(* CoDeSys 2.3.9.41 project: plastic_molding.pro *)
(* Libraries: Standard.lib 4.10.05 11:14:46, IecSfc.lib 13.4.06 15:51:28, SYSLIBCALLBACK.LIB 26.9.08 16:43:52 *)

(* Task configuration *)
TASK NewTask (PRIORITY := 1); (* freewheeling *)
	VIS_PRG();
	PLC_PRG();
END_TASK

(* Global variable list: Global_Variables *)
VAR_GLOBAL (* 11 inputs and 20 outputs *)
	(* Inputs *)
		(* Push buttons: *)
		StartPB: BOOL;
		StopPB: BOOL;
		InterruptPB: BOOL;

		(* Sensors: *)
		Weight0S: BOOL;
		Weight1S: BOOL;
		ClosedDamperS: BOOL;
		OpenedDamperS: BOOL;
		TareS: BOOL;
		UpperTempS: BOOL;
		BottomTempS: BOOL;
		WorkingTempS: BOOL;

	(* Outputs *)
		(* Actuators / Lamps *)
		StartFeed: BOOL;
		OpenValve: BOOL;
		RunConveyor: BOOL;
		OpenDamper: BOOL;
		CloseDamper: BOOL;
		TurnOnHeater: BOOL;

		(* States / Lamps *)
		SystemIsOn: BOOL;
		Stopping: BOOL;
		Melting: BOOL;
		NoFeed: BOOL;
		BrokenHeater: BOOL;
		NoTare: BOOL;

		(* Lamps *)
		EmptyDispenserLmp: BOOL;
		FullDispenserLmp: BOOL;
		TrippedTareSLmp: BOOL;
		OpenedDamperLmp: BOOL;
		ClosedDamperLmp: BOOL;
		UpperTempLmp: BOOL;
		BottomTempLmp: BOOL;
		WorkingTempLmp: BOOL;

	(* Timers are in global variables temporarily for convenience. *)
	FeederTmr: TON := (PT := T#7s);  (* Wating for feeding *)
	HeaterTmr: TON := (PT := T#12s); (* Wating for heating *)
	TareTmr: TON := (PT := T#7s); (* Waiting for tare *)
	MeltingTmr: TON := (PT := T#7s); (* Wating for melting *)
END_VAR

(* POU VIS_PRG, ST *)
PROGRAM VIS_PRG
VAR
	(* Buttons *)
	FillFeedingTowerBtn: BOOL;
	FreeFeedingTowerBtn: BOOL;
	HeaterBreakingToggleBtn: BOOL;
	FirstTareBtn, SecondTareBtn, ThirdTareBtn, FourthTareBtn  : BOOL;
	(* Others *)
	RawPlasticsVlm, _RawPlasticsVlm: INT;   (* Volume *)
	PlasticsPortionVlm,   _PlasticsPortionVlm: INT;  (* Volume *)
	PlasticsPortionClr:      DWORD;            (* Color *)
	Red,  _Red: INT;             (* Red component of the portion color *)
	(* Heater *)
	HeaterClr: DWORD:=16#00_FF_FF_FF;
	HeaterRed, _HeaterRed: BYTE;         (* Red component of the heater color  *)
	HeaterOn: BOOL;
	(* Conveyor *)
	ConveyorWheelsAngle: INT;
	_FirstTareShift: INT := -340;
	FirstTareShift: INT;
	_SecondTareShift: INT := -170;
	SecondTareShift: INT;
	_ThirsTareShift: INT := 0;
	ThirsTareShift: INT;
	_FourthTareShift : INT:= 170;
	FourthTareShift : INT;
	FirstTareVlm,   _FirstTareVlm, SecondTareVlm,   _SecondTareVlm, ThirdTareVlm,   _ThirdTareVlm,  FourthTareVlm,   _FourthTareVlm: INT;
	FirstTareVsb, SecondTareVsb, ThirsTareVsb, FourthTareVsb  : BOOL;
	(* Damper *)
	DamperShift: INT := 0;
	_DamperShift : INT;
END_VAR
(* Plastic volumes *)
RawPlasticsVlm := MAX(0, MIN(700,
		  BOOL_TO_INT(NOT FreeFeedingTowerBtn) * _RawPlasticsVlm + BOOL_TO_INT(FillFeedingTowerBtn) * 700 - BOOL_TO_INT(StartFeed)));
PlasticsPortionVlm :=  MAX(0, _PlasticsPortionVlm
				             +BOOL_TO_INT(StartFeed AND _RawPlasticsVlm > 0)
				             -BOOL_TO_INT(OpenValve AND _PlasticsPortionVlm  > 0) );
IF PlasticsPortionVlm = 0 THEN
	_Red := 0;
END_IF
Red := _Red + 2 * BOOL_TO_INT(ClosedDamperS AND NOT OpenValve) * (BOOL_TO_INT( _HeaterRed  >= 150) - BOOL_TO_INT( _HeaterRed < 150 AND _RED > 0));
PlasticsPortionClr := 65536*REAL_TO_BYTE(255 - Red)+REAL_TO_BYTE(Red);

(* Heater *)
HeaterOn:=TurnOnHeater AND NOT HeaterBreakingToggleBtn; (* Heater turn on if it is not broken  *)
HeaterRed:= _HeaterRed + BOOL_TO_BYTE(HeaterOn AND _HeaterRed < 255) - BOOL_TO_BYTE(NOT HeaterOn AND _HeaterRed > 0);
HeaterClr:=65536*(255 - HeaterRed)+256*(255 - HeaterRed)+255;

 (* Conveyor *)
ConveyorWheelsAngle := TIME_TO_INT(TareTmr.ET)/10;
FirstTareShift := (_FirstTareShift - BOOL_TO_INT(RunConveyor)*2 - 150) MOD 680 + 150;
SecondTareShift := (_SecondTareShift - BOOL_TO_INT(RunConveyor)*2 - 150) MOD 680 + 150;
ThirsTareShift := (_ThirsTareShift - BOOL_TO_INT(RunConveyor)*2 - 150) MOD 680 + 150;
FourthTareShift := (_FourthTareShift - BOOL_TO_INT(RunConveyor)*2 - 150) MOD 680 + 150;
FirstTareVsb := FirstTareShift > 0 OR FirstTareShift < -680 OR FirstTareBtn;
SecondTareVsb := SecondTareShift > 0 OR SecondTareShift < -680 OR SecondTareBtn ;
ThirsTareVsb := ThirsTareShift > 0 OR ThirsTareShift < -680 OR ThirdTareBtn;
FourthTareVsb := FourthTareShift > 0 OR FourthTareShift < -680 OR FourthTareBtn ;
IF FirstTareShift > 0 THEN
	FirstTareBtn := FALSE;
END_IF
IF SecondTareShift > 0 THEN
	SecondTareBtn := FALSE;
END_IF
IF ThirsTareShift > 0 THEN
	ThirdTareBtn := FALSE;
END_IF
IF FourthTareShift > 0 THEN
	FourthTareBtn := FALSE;
END_IF

(* Damper *)
DamperShift := _DamperShift - BOOL_TO_INT(CloseDamper) + BOOL_TO_INT(OpenDamper);


(* Sensors initialization *)
Weight0S := (PlasticsPortionVlm > 0);
Weight1S := (PlasticsPortionVlm = 40);
UpperTempS := (HeaterRed>=252);
BottomTempS := (HeaterRed>=160);
WorkingTempS := (HeaterRed>=150);
TareS := (FirstTareShift = -400 AND NOT FirstTareVsb) OR (SecondTareShift = -400 AND NOT SecondTareVsb) OR
		   (ThirsTareShift = -400 AND NOT ThirsTareVsb) OR (FourthTareShift = -400 AND NOT FourthTareVsb);
OpenedDamperS := DamperShift = 0;
ClosedDamperS := DamperShift = -50;

_RawPlasticsVlm := RawPlasticsVlm; _PlasticsPortionVlm := PlasticsPortionVlm; _Red := Red; _HeaterRed := HeaterRed; _FirstTareShift := FirstTareShift; _SecondTareShift := SecondTareShift;
_ThirsTareShift := ThirsTareShift; _FourthTareShift := FourthTareShift; _DamperShift := DamperShift;
END_PROGRAM

(* POU PLC_PRG, ST *)
PROGRAM PLC_PRG
VAR
	_SmoothStopping: BOOL; (* smooth stopping flag *)
	(* Pseudo-operator variables *)
	_SystemIsOn, _StopPB, _Stopping: BOOL;
	_WorkingTempS: BOOL;
END_VAR
(* Timers *)
FeederTmr.IN := StartFeed AND NOT Weight1S;
FeederTmr();
TareTmr.IN := RunConveyor AND NOT TareS;
TareTmr();
HeaterTmr.IN := TurnOnHeater AND NOT WorkingTempS;
HeaterTmr();
MeltingTmr.IN := _SystemIsOn AND ClosedDamperS AND WorkingTempS;
MeltingTmr();
(* 6 *)
IF NOT _SystemIsOn AND StartPB AND NOT StopPB THEN
	SystemIsOn := 1;
ELSIF _SystemIsOn AND (StopPB OR _SmoothStopping) THEN
	SystemIsOn := 0;
END_IF
(* 7 *)
_SmoothStopping := _Stopping AND
	NOT StartFeed AND RunConveyor AND NOT OpenDamper AND NOT CloseDamper AND
	NOT OpenValve AND OpenedDamperS AND Weight0S AND
	NOT BrokenHeater AND NOT NoTare AND NOT NoFeed;
(* 8 *)
IF NOT _Stopping AND _SystemIsOn AND StopPB THEN
	Stopping := 1;
ELSIF NOT _SystemIsOn THEN
	Stopping := 0;
END_IF
(* 9 *)
IF FeederTmr.Q AND NOT Weight1S THEN
	NoFeed := 1;
ELSIF NOT _SystemIsOn OR Weight1S THEN
	NoFeed := 0;
END_IF
(* 10 *)
IF TareTmr.Q AND NOT TareS THEN
	NoTare := 1;
ELSIF NOT _SystemIsOn OR TareS THEN
	NoTare := 0;
END_IF
(* 11 *)
IF HeaterTmr.Q  OR HeaterTmr.IN AND  _WorkingTempS THEN
	BrokenHeater := 1;
ELSIF NOT _SystemIsOn OR WorkingTempS THEN
	BrokenHeater := 0;
END_IF
(* 12 *)
StartFeed := _SystemIsOn AND OpenedDamperS AND
	(Weight0S AND NOT Weight1S OR NOT Weight0S AND NOT _SmoothStopping) AND
	NOT NoFeed;
(* 13 *)
OpenValve :=_SystemIsOn AND ClosedDamperS AND Weight0S AND TareS AND
	WorkingTempS AND MeltingTmr.Q AND
	NOT RunConveyor AND
	(Weight1S AND TareS OR OpenValve);
(* 14 *)
RunConveyor := _SystemIsOn AND NOT OpenValve AND
	(NOT TareS AND NOT NoTare OR TareS AND OpenValve);
(* 15 *)
CloseDamper :=_SystemIsOn AND Weight1S AND NOT ClosedDamperS;
(* 16 *)
OpenDamper :=_SystemIsOn AND NOT OpenValve AND NOT Weight1S AND NOT OpenedDamperS;
(* 17 *)
IF _SystemIsOn AND NOT BottomTempS AND NOT BrokenHeater AND NOT NoTare THEN
	TurnOnHeater := 1;
ELSIF NOT _SystemIsOn OR UpperTempS OR BrokenHeater OR NoTare THEN
	TurnOnHeater := 0;
END_IF
(* Lamps *)
EmptyDispenserLmp := Weight0S;
FullDispenserLmp := Weight1S;
TrippedTareSLmp := TareS;
OpenedDamperLmp := OpenedDamperS;
ClosedDamperLmp := ClosedDamperS;
UpperTempLmp := UpperTempS;
BottomTempLmp := BottomTempS;
WorkingTempLmp := WorkingTempS;
(* Pseudo-operator assignment *)
_SystemIsOn := SystemIsOn;
_StopPB := StopPB;
_Stopping := Stopping;
_WorkingTempS := WorkingTempS;
END_PROGRAM

(* Visualisation Plastic_molding
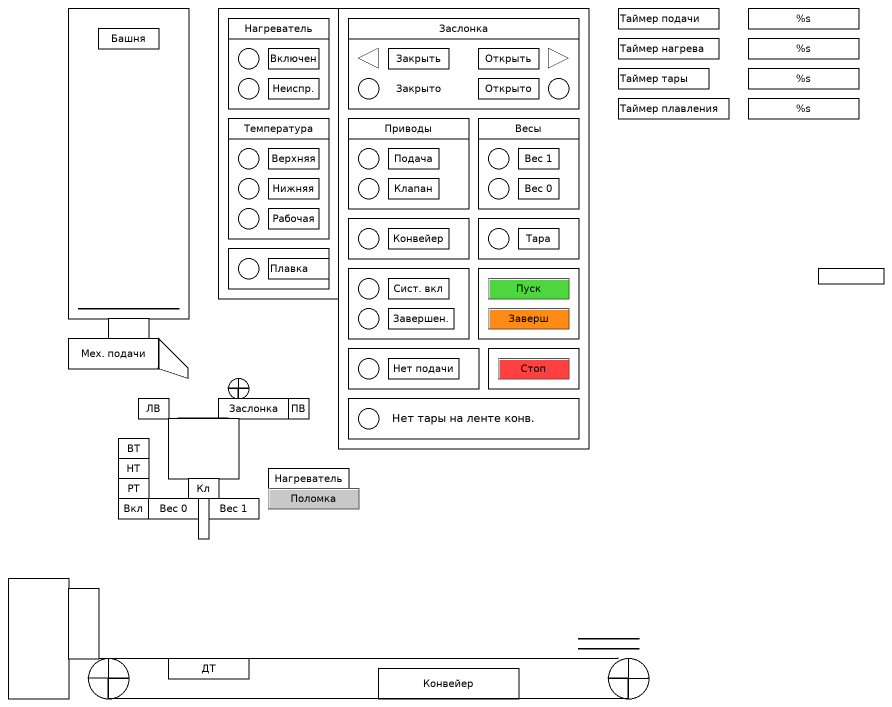
rectangle at (370,430)-(601,471): text "Нет тары на ленте конв."
ellipse at (380,440)-(401,461): alarm colour if .NoTare
ellipse at (380,390)-(401,411): alarm colour if .NoFeed
button at (520,390)-(591,411): text "Стоп"; taps .InterruptPB
button at (510,310)-(591,331): text "Пуск"; taps .StartPB
button at (510,340)-(591,361): text "Заверш"; taps .StopPB
ellipse at (510,260)-(531,281): alarm colour if .TrippedTareSLmp
rectangle at (370,150)-(491,171): text "Приводы"
rectangle at (500,150)-(601,171): text "Весы"
ellipse at (380,180)-(401,201): alarm colour if .StartFeed
ellipse at (380,210)-(401,231): alarm colour if .OpenValve
ellipse at (510,180)-(531,201): alarm colour if .FullDispenserLmp
ellipse at (510,210)-(531,231): alarm colour if .EmptyDispenserLmp
ellipse at (380,110)-(401,131): alarm colour if .ClosedDamperLmp
ellipse at (570,110)-(591,131): alarm colour if .OpenedDamperLmp
rectangle at (410,110)-(471,131): text "Закрыто"
rectangle at (500,110)-(561,131): text "Открыто"
rectangle at (410,180)-(461,201): text "Подача"
rectangle at (410,210)-(461,231): text "Клапан"
rectangle at (540,180)-(581,201): text "Вес 1"
rectangle at (540,210)-(581,231): text "Вес 0"
ellipse at (380,260)-(401,281): alarm colour if .RunConveyor
rectangle at (410,80)-(471,101): text "Закрыть"
polygon at (380,80)-(400,100): alarm colour if .CloseDamper
polygon at (570,80)-(590,100): alarm colour if .OpenDamper
rectangle at (500,80)-(561,101): text "Открыть"
rectangle at (370,50)-(601,71): text "Заслонка"
rectangle at (250,50)-(351,71): text "Нагреватель"
ellipse at (260,80)-(281,101): alarm colour if .TurnOnHeater
ellipse at (260,110)-(281,131): alarm colour if .BrokenHeater
rectangle at (290,80)-(341,101): text "Включен"
rectangle at (290,110)-(341,131): text "Неиспр."
rectangle at (250,150)-(351,171): text "Температура"
ellipse at (260,180)-(281,201): alarm colour if .UpperTempLmp
ellipse at (260,210)-(281,231): alarm colour if .BottomTempLmp
ellipse at (260,240)-(281,261): alarm colour if .WorkingTempLmp
rectangle at (290,180)-(341,201): text "Верхняя"
rectangle at (290,210)-(341,231): text "Нижняя"
rectangle at (290,240)-(341,261): text "Рабочая"
ellipse at (260,290)-(281,311): alarm colour if .Melting
rectangle at (290,290)-(351,311): text "Плавка"
rounded rectangle at (90,40)-(211,351): taps VIS_PRG.FillFeedingTowerBtn
rectangle at (100,340)-(201,341): taps VIS_PRG.FreeFeedingTowerBtn; top -VIS_PRG.RawPlasticsVlm/3
rectangle at (120,60)-(181,81): text "Башня"
rounded rectangle at (90,370)-(181,401): text "Мех. подачи"
rectangle at (240,430)-(311,451): text "Заслонка"; x offset VIS_PRG.DamperShift
rectangle at (310,430)-(331,451): text "ПВ"; alarm colour if .OpenedDamperS
rectangle at (160,430)-(191,451): text "ЛВ"; alarm colour if .ClosedDamperS
rectangle at (290,500)-(371,521): text "Нагреватель"
rectangle at (210,510)-(241,531): text "Кл"; alarm colour if .OpenValve
rectangle at (140,470)-(171,491): text "ВТ"; alarm colour if .UpperTempS
rectangle at (140,490)-(171,511): text "НТ"; alarm colour if .BottomTempS
rectangle at (140,510)-(171,531): text "РТ"; alarm colour if .WorkingTempS
rectangle at (140,530)-(171,551): text "Вкл"; alarm colour if .TurnOnHeater
rectangle at (170,530)-(221,551): text "Вес 0"; alarm colour if .Weight0S
rectangle at (230,530)-(281,551): text "Вес 1"; alarm colour if .Weight1S
polyline at (110,690)-(150,730): angle -VIS_PRG.ConveyorWheelsAngle
rectangle at (190,690)-(271,711): text "ДТ"; alarm colour if .TareS
polyline at (630,690)-(670,730): angle -VIS_PRG.ConveyorWheelsAngle
rectangle at (400,700)-(541,731): text "Конвейер"
ellipse at (380,310)-(401,331): alarm colour if .SystemIsOn
ellipse at (380,340)-(401,361): alarm colour if .Stopping
rectangle at (410,310)-(471,331): text "Сист. вкл"
rectangle at (410,340)-(476,361): text "Завершен."
rectangle at (410,390)-(481,411): text "Нет подачи"
rectangle at (410,260)-(471,281): text "Конвейер"
rectangle at (540,260)-(581,281): text "Тара"
rectangle at (640,40)-(741,61): text "Таймер подачи"
rectangle at (770,40)-(881,61): text "%s"; shows .FeederTmr.ET
rectangle at (770,70)-(881,91): text "%s"; shows .HeaterTmr.ET
rectangle at (640,70)-(741,91): text "Таймер нагрева"
rectangle at (640,100)-(731,121): text "Таймер тары"
rectangle at (640,130)-(751,151): text "Таймер плавления"
rectangle at (770,100)-(881,121): text "%s"; shows .TareTmr.ET
rectangle at (770,130)-(881,151): text "%s"; shows .MeltingTmr.ET
button at (290,520)-(381,541): text "Поломка"; toggles VIS_PRG.HeaterBreakingToggleBtn
rectangle at (600,680)-(661,681): invisible if VIS_PRG.FourthTareVsb; top -VIS_PRG.FourthTareVlm; x offset VIS_PRG.FourthTareShift
rectangle at (600,680)-(661,681): invisible if VIS_PRG.ThirsTareVsb; x offset VIS_PRG.ThirsTareShift
rectangle at (600,680)-(661,681): invisible if VIS_PRG.SecondTareVsb; top -VIS_PRG.SecondTareVlm; x offset VIS_PRG.SecondTareShift
rectangle at (600,680)-(661,681): invisible if VIS_PRG.FirstTareVsb; top -VIS_PRG.FirstTareVlm; x offset VIS_PRG.FirstTareShift
31 more shapes without text or variables
6 elements of other kinds (tables, trends, ...) not read
*)
